(* PLC project 6229, Phoenix Contact PC WORX 6.30 *)
(* stored: companyURL https://www.phoenixcontact-software.com, productRelease Build 593, creationDateTime 2020-08-26T14:19:07, contentDescription ###XMLINFO=2;1;2;;, version 0.1.240, modificationDateTime 2020-08-26T14:19:07 *)

FUNCTION_BLOCK SBT_DiagInfo_AddCRLF
  VAR_INPUT
    DiagInfo_In : SBT_V3_ARR_DIAG_INFO;
  END_VAR
  VAR_OUTPUT
    DiagInfo_Out : SBT_V3_ARR_DIAG_INFO;
  END_VAR
  VAR
    sTmp : SBT_V3_STR_400;
    sRet : SBT_V3_STR_400;
    i : INT;
    iPos : INT;
  END_VAR

						
							
								
							
							
								FOR i := 0 TO 16 BY 1 DO
	sTmp := DiagInfo_In[i];
	sRet := '';
	IF LEN(sTmp) > 0 THEN
		WHILE LEN(sTmp) > 70 DO
			sRet := CONCAT(sRet, LEFT(sTmp, 70));
		   	sTmp := DELETE(sTmp, 70, 1);
		   	iPos := FIND(sTmp, ' ');
		   	IF iPos > 0 THEN
		   		sRet := CONCAT(sRet, LEFT(sTmp, iPos));
				sRet := CONCAT(sRet, BYTE_TO_STRING(BYTE#16#0D, '%c'));
				sRet := CONCAT(sRet, BYTE_TO_STRING(BYTE#16#0A, '%c'));
		   		sTmp := DELETE(sTmp, iPos, 1);
			END_IF;
		END_WHILE;
									
		IF LEN(sTmp) > 0 THEN
			sRet := CONCAT(sRet, sTmp);
		END_IF;
	END_IF;
	DiagInfo_Out[i] := sRet;
END_FOR;
								
							
						
					
END_FUNCTION_BLOCK

FUNCTION_BLOCK Temperatur
  VAR_INPUT
    IN : INT;
  END_VAR
  VAR_OUTPUT
    ERROR : BOOL;
    ERRCODE : WORD;
    STR : STRING(80);
  END_VAR
  VAR
    strTmp : STRING(80);
  END_VAR

						
							
								
							
							
								IF (INT_TO_WORD(IN) & WORD#16#F000) <> WORD#16#8000 THEN
	ERROR := FALSE;
	ERRCODE := WORD#0;
	strTmp := REAL_TO_STRING(INT_TO_REAL(IN) / REAL#10.0, '%.1f °C');
	strTmp := REPLACE(strTmp, ',', 1, FIND(strTmp, '.'));
ELSE
	ERROR := TRUE;
	ERRCODE := INT_TO_WORD(IN);
	strTmp := '-,- °C';
END_IF;
									
STR := strTmp;
								
							
						
					
END_FUNCTION_BLOCK

PROGRAM SBT_Islands
  VAR_EXTERNAL
    xSBTCommOK : BOOL;
    xSBTDevError : BOOL;
  END_VAR
  VAR
    udtSBT : SBT_V3_UDT_SBT_V2;
  END_VAR
  VAR_EXTERNAL
    arrSBTOnlCntrlBuf : SBT_V3_ARR_DW_0_175;
    arrSBTOnlValBuf : SBT_V3_ARR_W_0_175;
    LPSDO_Out : SBT_V3_ARR_W_0_23;
    LPSDO_In : SBT_V3_ARR_W_0_23;
    Dev1_In : SBT_V3_ARR_W_0_3;
    Dev1_Out : SBT_V3_ARR_W_0_3;
  END_VAR
  VAR
    dwAppAck : DWORD;
    dwAppDiag : DWORD;
    xOpAckReq : BOOL;
    xQuitErrorDev1 : BOOL;
    xQuitErrorLPSDO : BOOL;
  END_VAR
  VAR_EXTERNAL
    MASTER_DIAG_STATUS_REG_DTC : BOOL;  (* Diagnostic routine active *)
    MASTER_DIAG_STATUS_REG_RUN : BOOL;  (* Data transmission active *)
  END_VAR
  VAR
    arr_wSBTdiagCode : SBT_V3_ARR_W_0_16;
    wDiagCodeLPSDO : WORD;
    wDiagCodeDev1 : WORD;
  END_VAR
  VAR_EXTERNAL
    xEStop : BOOL;
    I_NotAus : BOOL;
    I_Zweihand : BOOL;
  END_VAR
  VAR
    CLOCK_PULSE_1 : CLOCK_PULSE;
    SBT_V3_IBS_Restart_2_1 : SBT_V3_IBS_Restart_2;
    SBT_V3_BinFile_4_1 : SBT_V3_BinFile_4;
    SBT_V3_DiagCode_4_1 : SBT_V3_DiagCode_4;
    SBT_V3_OutBuff_4_1 : SBT_V3_OutBuff_4;
    SBT_V3_Operate_4_1 : SBT_V3_Operate_4;
    udtProjHeader : UDT_SBT_PROJ_HEADER;
    wAckDevErr : WORD;
    xAckOpErr : BOOL;
    xOpAckErr : BOOL;
    SBT_V3_InBuff_4_1 : SBT_V3_InBuff_4;
  END_VAR
  VAR_EXTERNAL
    xReset : BOOL;
  END_VAR
  VAR
    SBT_V3_DiagInfo_DE_1_1 : SBT_V3_DiagInfo_DE_1;
    arr_strSBTDiagInfo : SBT_V3_ARR_DIAG_INFO;
    SBT_DiagInfo_AddCRLF_1 : SBT_DiagInfo_AddCRLF;
    arr_strSBTDiagInfo2 : SBT_V3_ARR_DIAG_INFO;
    xError : BOOL;
    iDownload : INT;
    xDiffLogicDetected : BOOL;
    xAcceptDiffLogic : BOOL;
  END_VAR
  VAR_EXTERNAL
    xSBTDev1_CommOK : BOOL;
    xSBTLogicRunning : BOOL;
    xSBTReset : BOOL;
    I_Reset : BOOL;
  END_VAR
  VAR
    SBT_V3_ProjHeader_4_1 : SBT_V3_ProjHeader_4;
  END_VAR

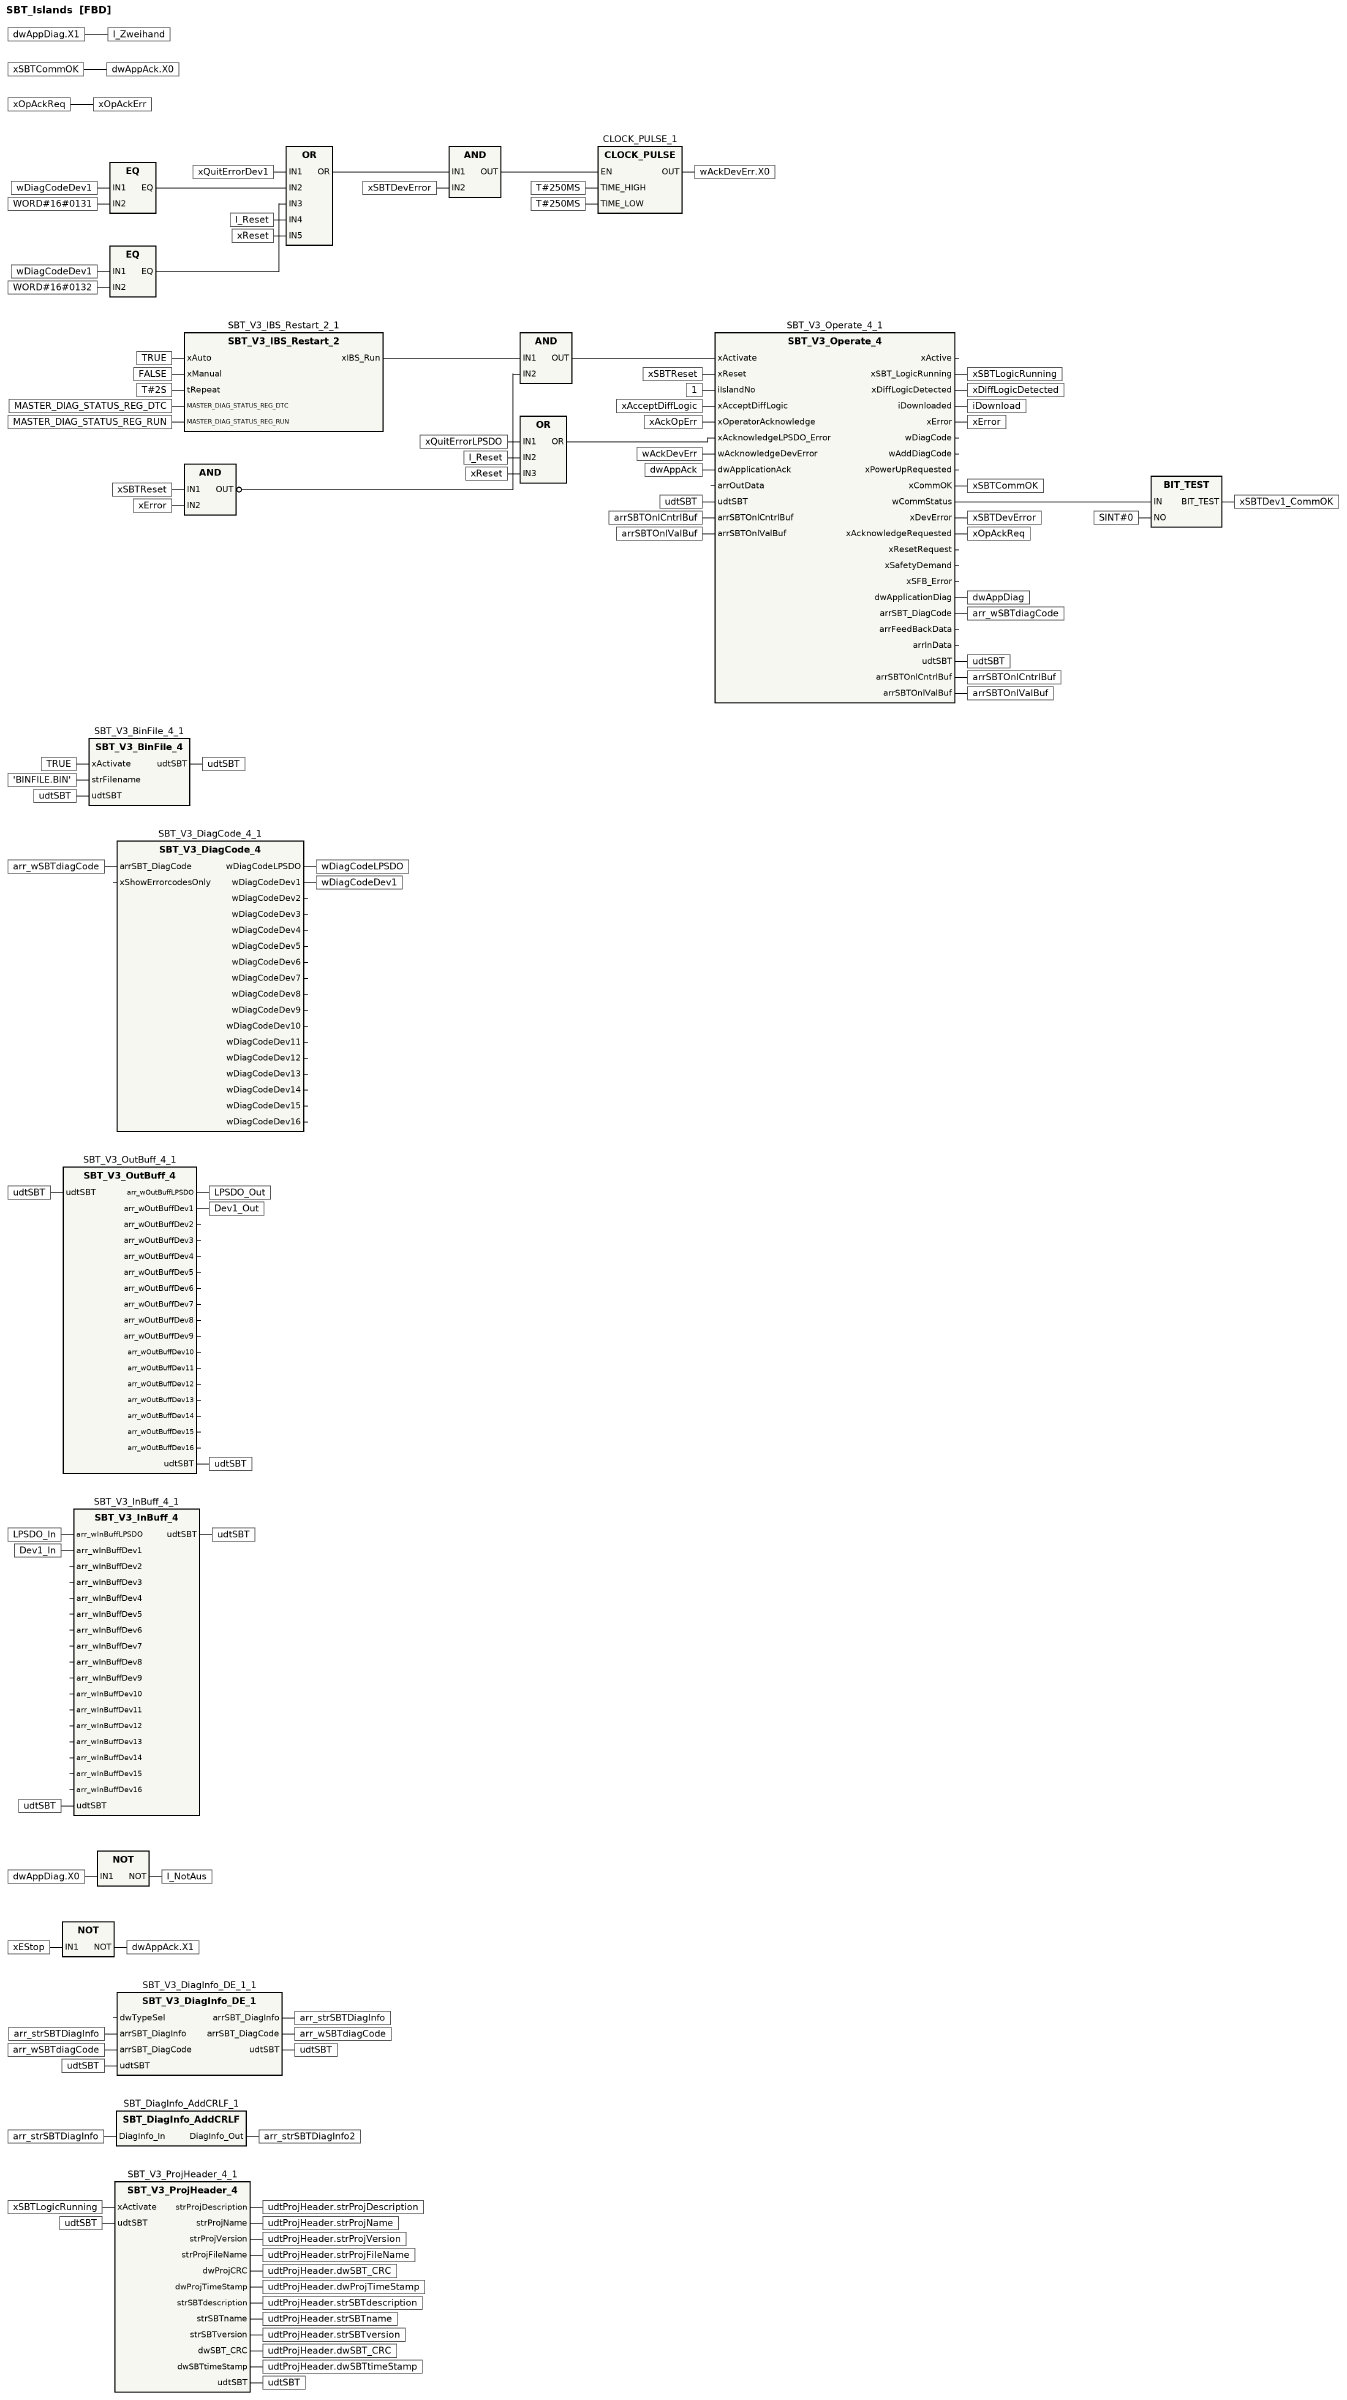
(* FBD diagram, written out as Structured Text *)
SBT_V3_BinFile_4_1(xActivate := TRUE, strFilename := 'BINFILE.BIN', udtSBT := udtSBT);
udtSBT := SBT_V3_BinFile_4_1.udtSBT;
SBT_V3_DiagCode_4_1(arrSBT_DiagCode := arr_wSBTdiagCode);
wDiagCodeLPSDO := SBT_V3_DiagCode_4_1.wDiagCodeLPSDO;
wDiagCodeDev1 := SBT_V3_DiagCode_4_1.wDiagCodeDev1;
SBT_V3_IBS_Restart_2_1(xAuto := TRUE, xManual := FALSE, tRepeat := T#2S, MASTER_DIAG_STATUS_REG_DTC := MASTER_DIAG_STATUS_REG_DTC, MASTER_DIAG_STATUS_REG_RUN := MASTER_DIAG_STATUS_REG_RUN);
SBT_V3_Operate_4_1(xActivate := SBT_V3_IBS_Restart_2_1.xIBS_Run AND NOT (xSBTReset AND xError), xReset := xSBTReset, iIslandNo := 1, xAcceptDiffLogic := xAcceptDiffLogic, xOperatorAcknowledge := xAckOpErr, xAcknowledgeLPSDO_Error := xQuitErrorLPSDO OR I_Reset OR xReset, wAcknowledgeDevError := wAckDevErr, dwApplicationAck := dwAppAck, udtSBT := udtSBT, arrSBTOnlCntrlBuf := arrSBTOnlCntrlBuf, arrSBTOnlValBuf := arrSBTOnlValBuf);
xDiffLogicDetected := SBT_V3_Operate_4_1.xDiffLogicDetected;
xSBTLogicRunning := SBT_V3_Operate_4_1.xSBT_LogicRunning;
SBT_V3_OutBuff_4_1(udtSBT := udtSBT);
LPSDO_Out := SBT_V3_OutBuff_4_1.arr_wOutBuffLPSDO;
xError := SBT_V3_Operate_4_1.xError;
iDownload := SBT_V3_Operate_4_1.iDownloaded;
Dev1_Out := SBT_V3_OutBuff_4_1.arr_wOutBuffDev1;
xSBTCommOK := SBT_V3_Operate_4_1.xCommOK;
xSBTDevError := SBT_V3_Operate_4_1.xDevError;
xOpAckReq := SBT_V3_Operate_4_1.xAcknowledgeRequested;
xSBTDev1_CommOK := BIT_TEST(SBT_V3_Operate_4_1.wCommStatus, SINT#0);
dwAppDiag := SBT_V3_Operate_4_1.dwApplicationDiag;
arr_wSBTdiagCode := SBT_V3_Operate_4_1.arrSBT_DiagCode;
SBT_V3_DiagInfo_DE_1_1(arrSBT_DiagInfo := arr_strSBTDiagInfo, arrSBT_DiagCode := arr_wSBTdiagCode, udtSBT := udtSBT);
arr_wSBTdiagCode := SBT_V3_DiagInfo_DE_1_1.arrSBT_DiagCode;
udtSBT := SBT_V3_DiagInfo_DE_1_1.udtSBT;
arr_strSBTDiagInfo := SBT_V3_DiagInfo_DE_1_1.arrSBT_DiagInfo;
SBT_V3_InBuff_4_1(arr_wInBuffLPSDO := LPSDO_In, arr_wInBuffDev1 := Dev1_In, udtSBT := udtSBT);
udtSBT := SBT_V3_InBuff_4_1.udtSBT;
arrSBTOnlCntrlBuf := SBT_V3_Operate_4_1.arrSBTOnlCntrlBuf;
udtSBT := SBT_V3_OutBuff_4_1.udtSBT;
arrSBTOnlValBuf := SBT_V3_Operate_4_1.arrSBTOnlValBuf;
udtSBT := SBT_V3_Operate_4_1.udtSBT;
SBT_DiagInfo_AddCRLF_1(DiagInfo_In := arr_strSBTDiagInfo);
arr_strSBTDiagInfo2 := SBT_DiagInfo_AddCRLF_1.DiagInfo_Out;
dwAppAck.X0 := xSBTCommOK;
dwAppAck.X1 := NOT xEStop;
I_Zweihand := dwAppDiag.X1;
I_NotAus := NOT dwAppDiag.X0;
SBT_V3_ProjHeader_4_1(xActivate := xSBTLogicRunning, udtSBT := udtSBT);
udtProjHeader.strProjDescription := SBT_V3_ProjHeader_4_1.strProjDescription;
udtProjHeader.strProjName := SBT_V3_ProjHeader_4_1.strProjName;
udtProjHeader.strProjVersion := SBT_V3_ProjHeader_4_1.strProjVersion;
udtProjHeader.strProjFileName := SBT_V3_ProjHeader_4_1.strProjFileName;
udtProjHeader.dwSBT_CRC := SBT_V3_ProjHeader_4_1.dwProjCRC;
xOpAckErr := xOpAckReq;
udtProjHeader.dwProjTimeStamp := SBT_V3_ProjHeader_4_1.dwProjTimeStamp;
udtProjHeader.strSBTdescription := SBT_V3_ProjHeader_4_1.strSBTdescription;
udtProjHeader.strSBTname := SBT_V3_ProjHeader_4_1.strSBTname;
CLOCK_PULSE_1(EN := (xQuitErrorDev1 OR wDiagCodeDev1 = WORD#16#0131 OR wDiagCodeDev1 = WORD#16#0132 OR I_Reset OR xReset) AND xSBTDevError, TIME_HIGH := T#250MS, TIME_LOW := T#250MS);
IF CLOCK_PULSE_1.ENO THEN wAckDevErr.X0 := CLOCK_PULSE_1.OUT; END_IF;
udtProjHeader.strSBTversion := SBT_V3_ProjHeader_4_1.strSBTversion;
udtSBT := SBT_V3_ProjHeader_4_1.udtSBT;
udtProjHeader.dwSBT_CRC := SBT_V3_ProjHeader_4_1.dwSBT_CRC;
udtProjHeader.dwSBTtimeStamp := SBT_V3_ProjHeader_4_1.dwSBTtimeStamp;
END_PROGRAM

FUNCTION_BLOCK Automatik
  VAR
    iStep : INT;
  END_VAR
  VAR_EXTERNAL
    Q_ZylRechtsGs : BOOL;  (* Zylinder in Grundstellung *)
    Q_ZylRechtsAs : BOOL;  (* Zylinder in Arbeitsstellung *)
    Q_ZylLinksGs : BOOL;  (* Zylinder in Grundstellung *)
    Q_ZylLinksAs : BOOL;  (* Zylinder in Arbeitsstellung *)
    Q_DruckerStart : BOOL;
  END_VAR
  VAR
    R_TRIG_1 : R_TRIG;
  END_VAR
  VAR_EXTERNAL
    I_Zweihand : BOOL;
    I_TawGewBuchseLinks : BOOL;  (* Teilanwesenheit Gewindebuchse links *)
    I_TawGewBuchseRechts : BOOL;  (* Teilanwesenheit Gewindebuchse rechts *)
    I_TawLagerbuchseLinks : BOOL;  (* Teilanwesenheit Lagerbuchse links *)
    I_TawLagerbuchseRechts : BOOL;  (* Teilanwesenheit Lagerbuchse rechts *)
    I_ZylLinksGs : BOOL;  (* Zylinder links ist in Grundstellung *)
    I_ZylLinksAs : BOOL;  (* Zylinder links ist in Arbeitsstellung *)
    I_ZylRechtsGs : BOOL;  (* Zylinder rechts ist in Grundstellung *)
    I_DruckerBereit : BOOL;
    I_DruckerFehler : BOOL;
    I_NotAus : BOOL;
  END_VAR
  VAR
    TON_1 : TON;
  END_VAR
  VAR_EXTERNAL
    I_ZylRechtsAs : BOOL;  (* Zylinder rechts ist in Arbeitsstellung *)
    xStoerung : BOOL;
    I_DruckluftOK : BOOL;  (* Druckluft ist vorhanden *)
    I_Nachpressen : BOOL;
    xAuto : BOOL;
    xZuHeissOderDefekt : BOOL;
  END_VAR
  VAR
    xTeilOK : BOOL;
  END_VAR

						
							
								
							
							
								R_TRIG_1(CLK:=I_Zweihand);
TON_1(IN:=I_ZylLinksAs AND I_ZylRechtsAs,PT:=T#750MS);
									
IF NOT xAuto THEN
	RETURN;
END_IF;
									
IF I_NotAus OR xStoerung OR xZuHeissOderDefekt THEN
	Q_ZylLinksGs := xStoerung;
	Q_ZylLinksAs := FALSE;
	Q_ZylRechtsGs := xStoerung;
	Q_ZylRechtsAs := FALSE;
	Q_DruckerStart := FALSE;
	iStep := 0;
END_IF;
									
CASE iStep OF
	0:
		IF I_ZylLinksGs AND I_ZylRechtsGs THEN
			IF xTeilOK AND NOT I_TawLagerbuchseLinks AND NOT I_TawLagerbuchseRechts THEN
				Q_DruckerStart := Not I_Nachpressen;
			END_IF;
									
			xTeilOK := FALSE;
		END_IF;
									
		IF I_DruckluftOK AND R_TRIG_1.Q AND I_TawGewBuchseLinks AND I_TawGewBuchseRechts AND
		(I_TawLagerbuchseLinks Or (I_Nachpressen And Not I_TawLagerbuchseLinks)) AND
		(I_TawLagerbuchseRechts Or (I_Nachpressen And Not I_TawLagerbuchseRechts)) AND
		I_ZylLinksGs AND I_ZylRechtsGs AND ((I_DruckerBereit AND NOT I_DruckerFehler) Or I_Nachpressen) THEN
			Q_DruckerStart := FALSE;
			iStep := iStep + 1;
		END_IF;
									
		IF I_DruckluftOK AND R_TRIG_1.Q AND (NOT I_ZylLinksGs OR NOT I_ZylRechtsGs) THEN
			iStep := 100;
		END_IF;
									
	1:
		Q_ZylLinksAs := TRUE;
		Q_ZylRechtsAs := TRUE;
									
		IF TON_1.Q THEN
			xTeilOK := TRUE;
			Q_ZylLinksAs := FALSE;
			Q_ZylRechtsAs := FALSE;
			iStep := iStep + 1;
		END_IF;
									
	2:
		Q_ZylLinksGs := TRUE;
		Q_ZylRechtsGs := TRUE;
									
		IF I_ZylLinksGs AND I_ZylRechtsGs THEN
			Q_ZylLinksGs := FALSE;
			Q_ZylRechtsGs := FALSE;
			iStep := 0;
		END_IF;
									
	100:
		Q_ZylLinksAs := FALSE;
		Q_ZylLinksGs := TRUE;
		Q_ZylRechtsAs := FALSE;
		Q_ZylRechtsGs := TRUE;
									
		IF xTeilOK THEN
			xTeilOK := FALSE;
			Q_DruckerStart := Not I_Nachpressen;
		END_IF;
									
		IF I_ZylLinksGs AND I_ZylRechtsGs THEN
			Q_ZylLinksGs := FALSE;
			Q_ZylRechtsGs := FALSE;
			iStep := 0;
		END_IF;
END_CASE;
 
								
							
						
					
END_FUNCTION_BLOCK

PROGRAM Main
  VAR_EXTERNAL
    ONBOARD_OUTPUT_BIT0 : BOOL;  (* Local output OUT1 *)
    I_DruckluftOK : BOOL;  (* Druckluft ist vorhanden *)
    ONBOARD_INPUT_BIT3 : BOOL;  (* Local input IN4 *)
    ONBOARD_INPUT_BIT0 : BOOL;  (* Local input IN1 *)
    ONBOARD_INPUT_BIT1 : BOOL;  (* Local input IN2 *)
    I_DruckerBereit : BOOL;
    I_DruckerFehler : BOOL;
    Q_DruckerStart : BOOL;
    Q_ZylLinksAs : BOOL;  (* Zylinder in Arbeitsstellung *)
    Q_ZylLinksGs : BOOL;  (* Zylinder in Grundstellung *)
    I_Zweihand : BOOL;
    xEStop : BOOL;
    ONBOARD_INPUT_BIT4 : BOOL;  (* Local input IN5 *)
    Q_LmGruen : BOOL;  (* Leuchtmelder grün *)
    xSBTCommOK : BOOL;
    xSBTDevError : BOOL;
    I_NotAus : BOOL;
  END_VAR
  VAR
    TON_1 : TON;
  END_VAR
  VAR_EXTERNAL
    I_ZylLinksGs : BOOL;  (* Zylinder links ist in Grundstellung *)
    I_ZylRechtsGs : BOOL;  (* Zylinder rechts ist in Grundstellung *)
  END_VAR
  VAR
    SR_2 : SR;
  END_VAR
  VAR_EXTERNAL
    xStoerung : BOOL;
  END_VAR
  VAR
    TON_2 : TON;
  END_VAR
  VAR_EXTERNAL
    I_ZylLinksAs : BOOL;  (* Zylinder links ist in Arbeitsstellung *)
    I_ZylRechtsAs : BOOL;  (* Zylinder rechts ist in Arbeitsstellung *)
  END_VAR
  VAR
    CLOCK_PULSE_5 : CLOCK_PULSE;
  END_VAR
  VAR_EXTERNAL
    I_Reset : BOOL;
    ONBOARD_INPUT_BIT5 : BOOL;  (* Local input IN6 *)
    I_Nachpressen : BOOL;
    I_TemperaturLuft : INT;
    strTemperaturLuft : STRING(80);
    I_TemperaturTeil : INT;
    strTemperaturTeil : STRING(80);
  END_VAR
  VAR
    Temperatur_1 : Temperatur;
    Temperatur_2 : Temperatur;
  END_VAR
  VAR_EXTERNAL
    xAuto : BOOL;
  END_VAR
  VAR
    Automatik_1 : Automatik;
  END_VAR
  VAR_EXTERNAL
    ONBOARD_OUTPUT_BIT3 : BOOL;  (* Local output OUT4 *)
    Q_ZylRechtsGs : BOOL;  (* Zylinder in Grundstellung *)
    xReset : BOOL;
  END_VAR
  VAR
    SR_1 : SR;
  END_VAR
  VAR_EXTERNAL
    xSBTDev1_CommOK : BOOL;
    xSBTLogicRunning : BOOL;
    iMaxTemp : INT;
    xCheckTemp : BOOL;
  END_VAR
  VAR
    CLOCK_PULSE_1 : CLOCK_PULSE;
  END_VAR
  VAR_EXTERNAL
    xZuHeiss_Pulsed : BOOL;
    Q_ZylRechtsAs : BOOL;  (* Zylinder in Arbeitsstellung *)
    xZuHeissOderDefekt : BOOL;
  END_VAR
  VAR  (* added by the conversion: wires and edge detectors of the diagram *)
    _DIV321_OUT : REAL;
    _INT_TO_REAL325_OUT : REAL;
    _GT319_OUT : BOOL;
  END_VAR

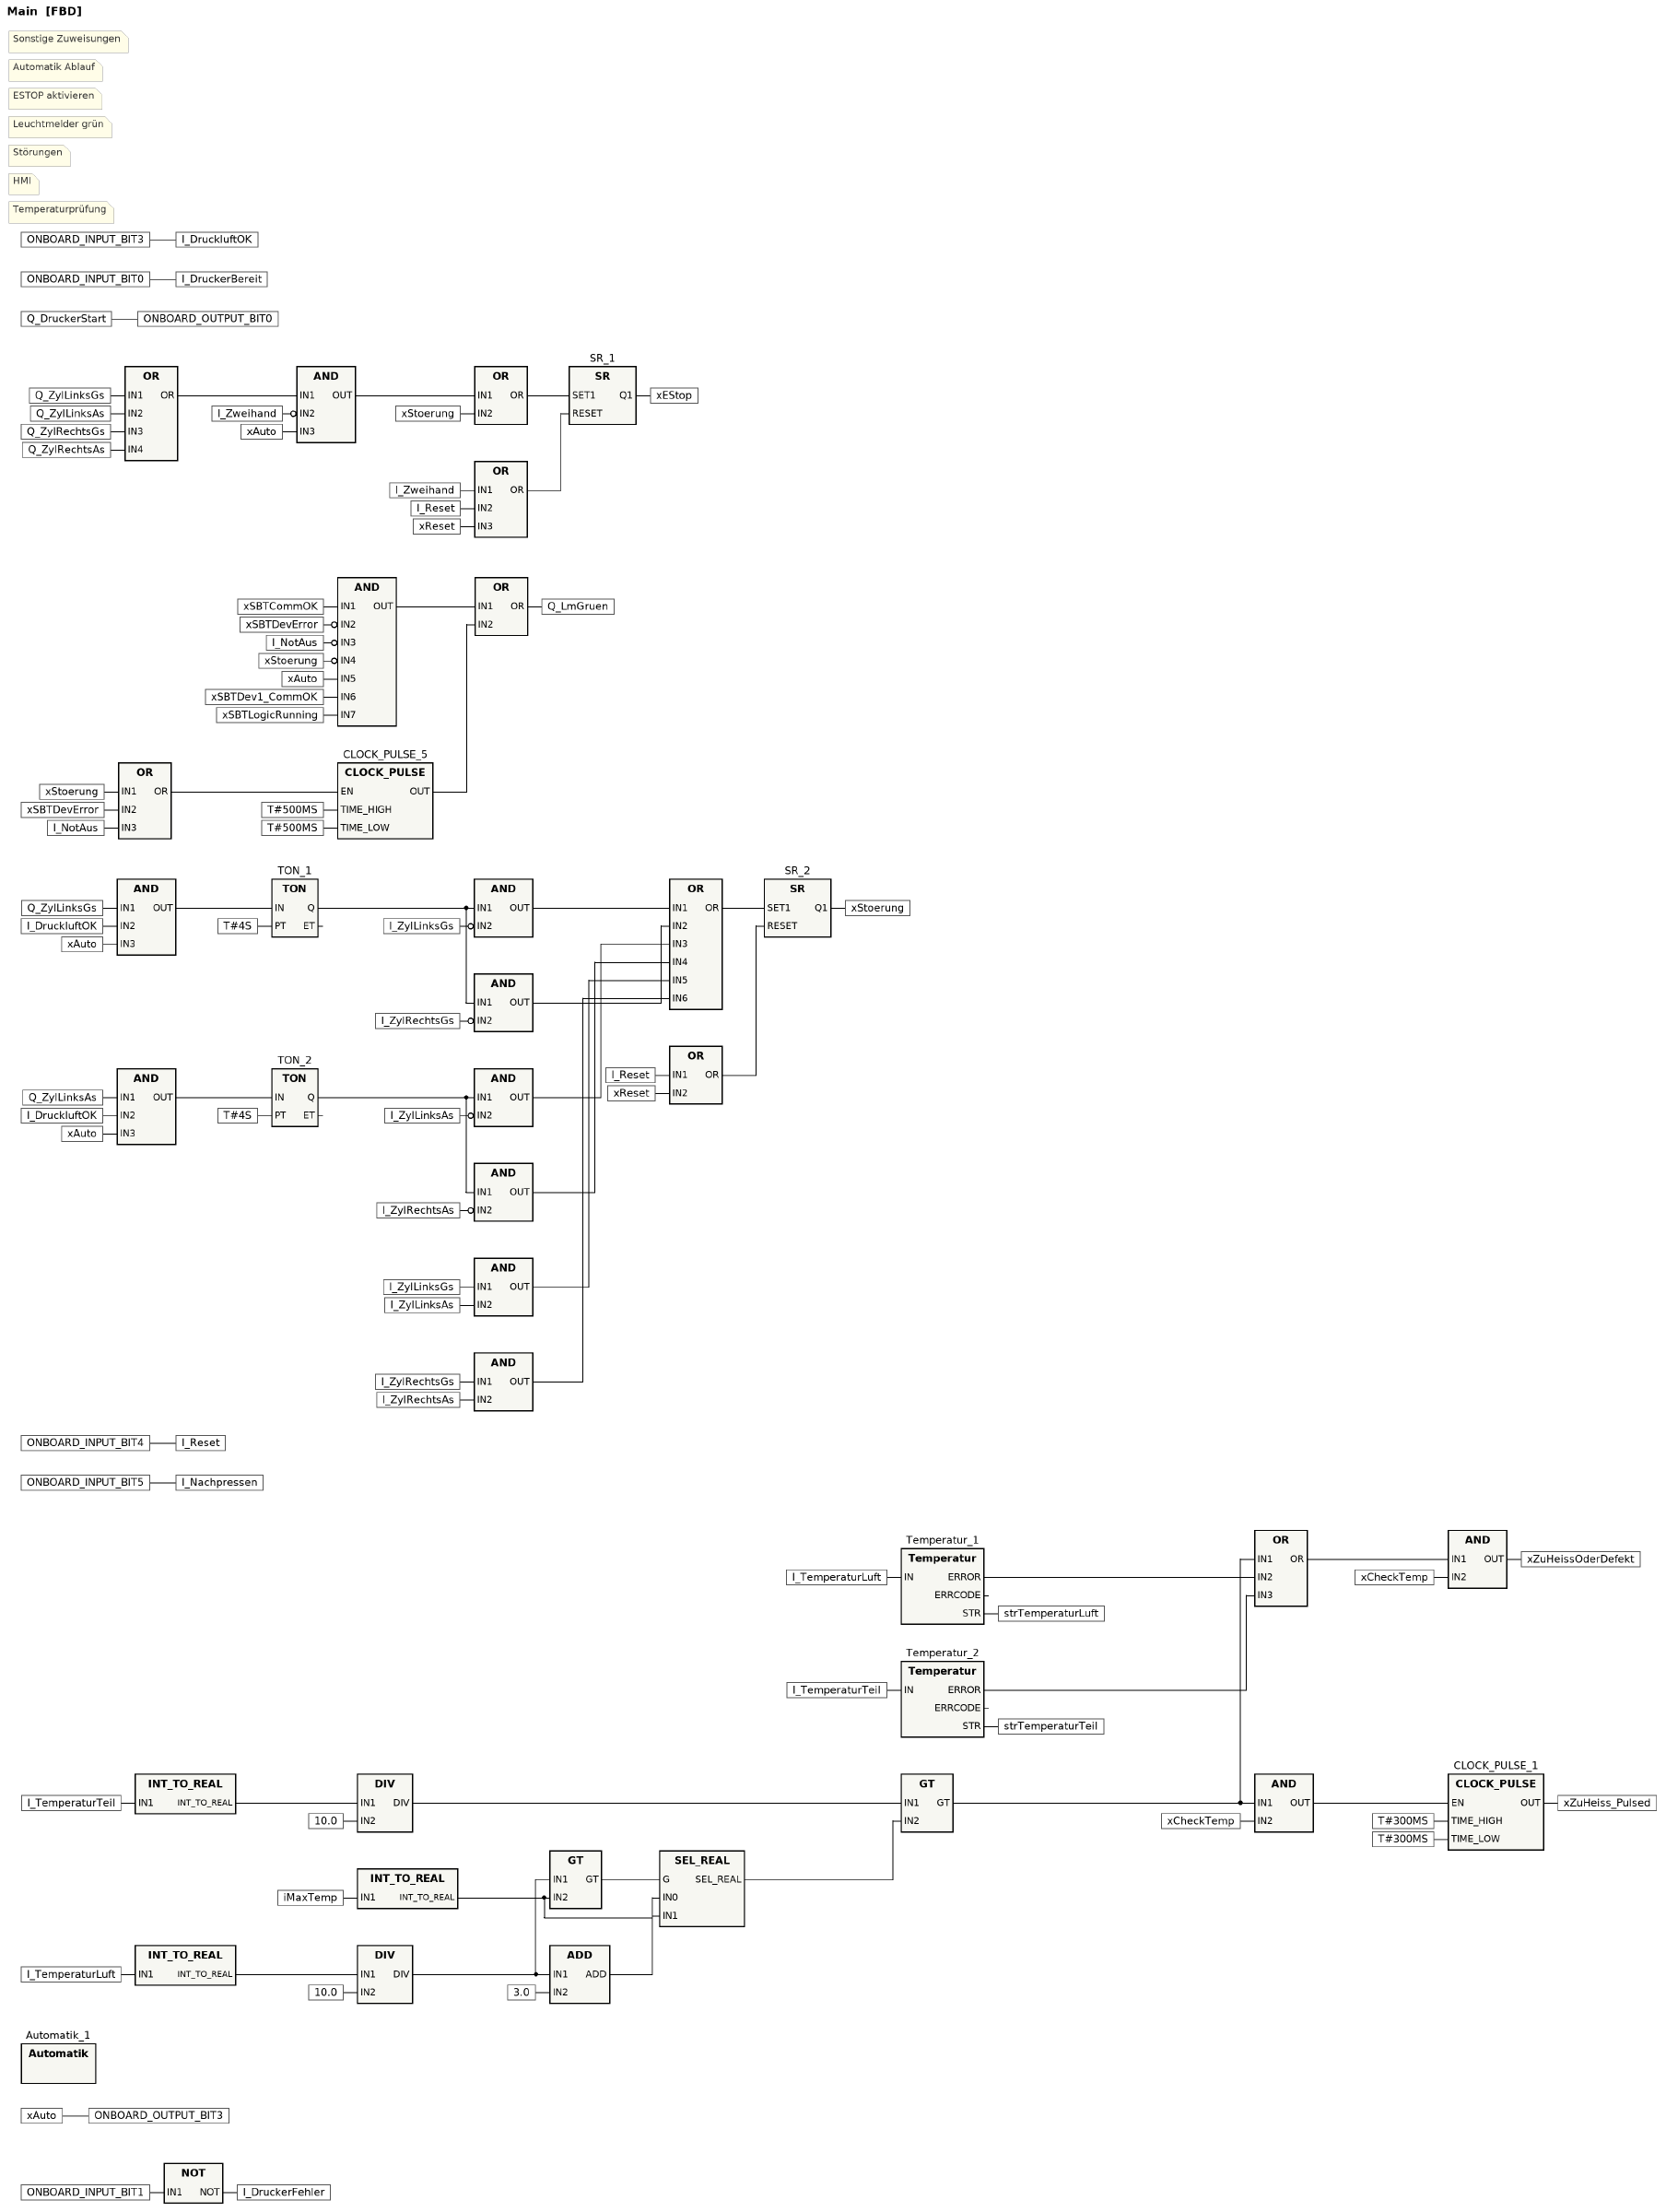
(* FBD diagram, written out as Structured Text *)
(* Automatik Ablauf *)
(* Sonstige Zuweisungen *)
(* ESTOP aktivieren *)
I_DruckerBereit := ONBOARD_INPUT_BIT0;
I_DruckluftOK := ONBOARD_INPUT_BIT3;
I_DruckerFehler := NOT ONBOARD_INPUT_BIT1;
ONBOARD_OUTPUT_BIT0 := Q_DruckerStart;
ONBOARD_OUTPUT_BIT3 := xAuto;
SR_1(SET1 := (Q_ZylLinksGs OR Q_ZylLinksAs OR Q_ZylRechtsGs OR Q_ZylRechtsAs) AND NOT I_Zweihand AND xAuto OR xStoerung, RESET := I_Zweihand OR I_Reset OR xReset);
xEStop := SR_1.Q1;
I_Reset := ONBOARD_INPUT_BIT4;
I_Nachpressen := ONBOARD_INPUT_BIT5;
(* Störungen *)
(* Leuchtmelder grün *)
TON_1(IN := Q_ZylLinksGs AND I_DruckluftOK AND xAuto, PT := T#4S);
TON_2(IN := Q_ZylLinksAs AND I_DruckluftOK AND xAuto, PT := T#4S);
SR_2(SET1 := TON_1.Q AND NOT I_ZylLinksGs OR TON_1.Q AND NOT I_ZylRechtsGs OR TON_2.Q AND NOT I_ZylLinksAs OR TON_2.Q AND NOT I_ZylRechtsAs OR I_ZylLinksGs AND I_ZylLinksAs OR I_ZylRechtsGs AND I_ZylRechtsAs, RESET := I_Reset OR xReset);
xStoerung := SR_2.Q1;
CLOCK_PULSE_5(EN := xStoerung OR xSBTDevError OR I_NotAus, TIME_HIGH := T#500MS, TIME_LOW := T#500MS);
Q_LmGruen := xSBTCommOK AND NOT xSBTDevError AND NOT I_NotAus AND NOT xStoerung AND xAuto AND xSBTDev1_CommOK AND xSBTLogicRunning OR CLOCK_PULSE_5.OUT;
(* HMI *)
(* Temperaturprüfung *)
Temperatur_1(IN := I_TemperaturLuft);
strTemperaturLuft := Temperatur_1.STR;
Temperatur_2(IN := I_TemperaturTeil);
strTemperaturTeil := Temperatur_2.STR;
_DIV321_OUT := INT_TO_REAL(I_TemperaturLuft) / 10.0;
_INT_TO_REAL325_OUT := INT_TO_REAL(iMaxTemp);
_GT319_OUT := INT_TO_REAL(I_TemperaturTeil) / 10.0 > SEL_REAL(_DIV321_OUT > _INT_TO_REAL325_OUT, _INT_TO_REAL325_OUT, _DIV321_OUT + 3.0);
xZuHeissOderDefekt := (_GT319_OUT OR Temperatur_1.ERROR OR Temperatur_2.ERROR) AND xCheckTemp;
CLOCK_PULSE_1(EN := _GT319_OUT AND xCheckTemp, TIME_HIGH := T#300MS, TIME_LOW := T#300MS);
IF CLOCK_PULSE_1.ENO THEN xZuHeiss_Pulsed := CLOCK_PULSE_1.OUT; END_IF;
Automatik_1();
END_PROGRAM
